(* CODESYS project FU_wBitPart.xml

Project tree, tasks and I/O mapping:
  function FU_wBitPart [ST]
*)

// FU_wBitPart
//This function changed only the needed bits of a variable
// |**Version**|**Author**| **Date** |**Changes**
// | 1         | NSN      | 16-03-22 | Creation
FUNCTION FU_wBitPart : BOOL
VAR_IN_OUT
	valueChange		:WORD;		//Variable to change
END_VAR
VAR_INPUT
	value			:WORD;		//Value to change bits to
	amount			:BYTE;		//Amount of bits to change
	offset			:BYTE;		//Offset in variable to change bits at
END_VAR

valueChange		:=		(valueChange AND ROL(GConstants.binaryInvMaskWord[amount],offset)) OR SHL(value AND GConstants.binaryMaskWord[amount],offset);

END_FUNCTION
